FUNCTION F_CallLogTask

GlobalVariables.aTaskLogger[GETCURTASKINDEXEX()].Call();

END_FUNCTION

(* stored: Version 1.1.0.1, ProductVersion 3.1.4024.0
   POU F_CallLogTask: Id {43b77b84-3ad4-4dba-a1e5-4c575f461237}, SpecialFunc None *)
